// TIA Portal V17 export
// export: Created 2024-08-07T21:44:09.0950211Z, ExportSetting WithDefaults, DisplayName Totally Integrated Automation Portal, DisplayVersion V17 Update 7, DisplayName TIA Portal Openness, DisplayVersion V17 Update 7, DisplayName TIA Portal Version Control Interface, DisplayVersion V17, DisplayName SINAMICS Startdrive Advanced, DisplayVersion V17 SP2, DisplayName SINAMICS Startdrive G110M, G120, G120C, G120D, G120P, G115D, DisplayVersion V17 SP2, DisplayName SINAMICS Startdrive G130, G150, S120, S150, SINAMICS MV, S210, DisplayVersion V17 SP2, DisplayName STEP 7 Professional, DisplayVersion V17 Update 7, DisplayName STEP 7 Safety, DisplayVersion V17 Update 6, DisplayName WinCC Advanced / Unified PC, DisplayVersion V17 Update 7
DATA_BLOCK "ValueContinuityCheck_VH2_DB"   // DB52
VERSION : 0.1
// stored: AutoNumber true, DBAccessibleFromOPCUA true, DBAccessibleFromWebserver true, InstanceOfName ValueContinuityCheck, InstanceOfType FB
"ValueContinuityCheck"
   // VAR_INPUT
   //    valueToCheck : Real;
   //    changeLimitForScan : Real;
   //    reset : Bool;
   // END_VAR
   // VAR_OUTPUT
   //    error : Bool;
   //    changeDuringError : Real;
   // END_VAR
   // VAR
   //    valueMemory : Real;
   //    biggestChange : Real;
   // END_VAR
BEGIN
END_DATA_BLOCK
